{attribute 'qualified_only'}
VAR_GLOBAL CONSTANT
    nSources : UINT := 8;
    (* Destinations

        LTLHN:LD2:VGC:01 (ioc-las-bts) - TMO - IP3
        LTLHN:LD4:VGC:01 (ioc-las-bts) - RIX - ChemRIXS
        LTLHN:LD6:VGC:01 (ioc-las-bts) - RIX - qRIXS
        LTLHN:LD8:VGC:01 (ioc-las-bts) - TMO - IP1
        LTLHN:LD9:VGC:01 (ioc-las-bts) - Laser Lab
        LTLHN:LD10:VGC:01 (ioc-las-bts) - TMO - IP2
        LTLHN:LD14:VGC:01 (ioc-las-bts) - XPP

    *)
    nDestinations: UINT := 14;
END_VAR

(* stored: Version 1.1.0.1, ProductVersion 3.1.4022.18
   GVL GVL_BTPS_Constants: Id {9a37ab9e-aa73-4851-ba45-23ade47dd444} *)
